{attribute 'strict'}
TYPE E_MachineCtrlStateUninitialized :
(	
	(*Robot uninitializing *)
	MACHINE_STATE_UNINITIALIZED_POWER_ON_CR800 						:= 0,	
	MACHINE_STATE_UNINITIALIZED_CR800_ETHERCAT_STATUS_CHECK 		:= 10,
	MACHINE_STATE_UNINITIALIZED_CR800_ETHERCAT_STATUS_CHECK_DONE	:= 20,
	MACHINE_STATE_UNINITIALIZED_CR800_ETHERCAT_ERROR_RESET			:= 30,
	MACHINE_STATE_UNINITIALIZED_CR800_ETHERCAT_REQUEST_OP_STATE		:= 40,	(*  *)	
	MACHINE_STATE_UNINITIALIZED_CR800_CHECK_POWER_REGISTER			:= 50,	(*  *)
	(* Vision *)
	
	(* Driver *)
	MACHINE_STATE_UNINITIALIZED_DRIVER_POWER_CHECK					:= 100,
	
	MACHINE_STATE_UNINITIALIZED_DONE								:= 200	(*  *)
);
END_TYPE

(* stored: Version 1.1.0.1, ProductVersion 3.1.4024.9
   DUT E_MachineCtrlStateUninitialized: Id {b9fdefb4-3200-4e13-b096-7e163c427a60} *)
